PROGRAM p_ModbusTx_PLCMemory
VAR
END_VAR

MEMCPY(destAddr:=ADR(mb_PLC_Memory[10]), srcAddr:=ADR(vgPBT_GCC_02.rPRESS), n:=SIZEOF(vgPBT_GCC_02.rPRESS));  //VG pressure readbacks
MEMCPY(destAddr:=ADR(mb_PLC_Memory[12]), srcAddr:=ADR(vgPBT_GCC_04.rPRESS), n:=SIZEOF(vgPBT_GCC_04.rPRESS));  //VG pressure readbacks
MEMCPY(destAddr:=ADR(mb_PLC_Memory[14]), srcAddr:=ADR(vgPBT_GCC_06.rPRESS), n:=SIZEOF(vgPBT_GCC_06.rPRESS));  //VG pressure readbacks
MEMCPY(destAddr:=ADR(mb_PLC_Memory[16]), srcAddr:=ADR(vgPBT_GCC_07.rPRESS), n:=SIZEOF(vgPBT_GCC_07.rPRESS));  //VG pressure readbacks
MEMCPY(destAddr:=ADR(mb_PLC_Memory[18]), srcAddr:=ADR(vgPBT_GCC_08.rPRESS), n:=SIZEOF(vgPBT_GCC_08.rPRESS));  //VG pressure readbacks

END_PROGRAM

(* stored: Version 1.1.0.1, ProductVersion 3.1.4020.12
   POU p_ModbusTx_PLCMemory: Id {1375f286-8a4d-4ae5-8ad4-ba6b3a50bbf6}, SpecialFunc None *)
